// TIA Portal V20 export
// export: Created 2026-10-03T18:54:34.7220554Z, ExportSetting WithDefaults, DisplayName Totally Integrated Automation Portal, DisplayVersion V20 Update 4, DisplayName TIA Portal Openness, DisplayVersion V20 Update 4, DisplayName TIA Portal Version Control Interface, DisplayVersion V20 Update 4, DisplayName SINAMICS Startdrive Advanced, DisplayVersion V20 SP1 Update 1, DisplayName SINAMICS Startdrive G110M, G120, G120C, G120D, G120P, G115D, DisplayVersion V20 SP1 Update 1, DisplayName SINAMICS Startdrive G130, G150, S120, S150, SINAMICS MV, G220, S200, S210, DisplayVersion V20 SP1 Update 1, DisplayName STEP 7 Professional, DisplayVersion V20 Update 4, DisplayName STEP 7 Safety, DisplayVersion V20 Update 2, DisplayName WinCC Basic/Comfort/Advanced, DisplayVersion V20 Update 4, DisplayName WinCC Unified, DisplayVersion V20 Update 4
FUNCTION "SLC_STATUS" : Void   // FC22, SCL
TITLE = SLC status file clocks
{ S7_Optimized_Access := 'TRUE' }
VERSION : 0.1
// Keeps the SLC status words that the logic reads as clocks up to date, so rungs such as XIC S:4/7 or NEQ S:42 N7:2
//  work exactly as in the SLC without any CPU settings. Called at the start of Main.
// stored: AutoNumber true, IsIECCheckEnabled false, SetENOAutomatically false, UDAEnableTagReadback false
   VAR_OUTPUT
      FreeRunningClock : Int;   // S:4: counts up every 10 ms and wraps at 16 bits, like the SLC's
      Year : Int;   // S:37
      Month : Int;   // S:38
      Day : Int;   // S:39
      Hour : Int;   // S:40
      Minute : Int;   // S:41
      Second : Int;   // S:42
   END_VAR
   VAR_TEMP
      now : DTL;
      status : Int;
   END_VAR
BEGIN
   // The CPU's millisecond tick counter, in 10 ms counts, keeping only the low 16 bits as the SLC does.
   #FreeRunningClock := WORD_TO_INT(DINT_TO_WORD(TIME_TO_DINT(TIME_TCK()) / 10));

   // The CPU's local date and time.
   #status := RD_LOC_T(#now);
   #Year := UINT_TO_INT(#now.YEAR);
   #Month := USINT_TO_INT(#now.MONTH);
   #Day := USINT_TO_INT(#now.DAY);
   #Hour := USINT_TO_INT(#now.HOUR);
   #Minute := USINT_TO_INT(#now.MINUTE);
   #Second := USINT_TO_INT(#now.SECOND);
END_FUNCTION
